TYPE "Positioning_MOL_Machine_Pers_Data"
VERSION : 0.1
// Block: Positioning_MOL_Machine_Pers_Data
   STRUCT
      AxisHomed : Bool;
   END_STRUCT;

END_TYPE
